FUNCTION_BLOCK farbzuordnung (* Basic Function Block Type *)
  (* Standard: 61499-2 *)
  (* Version 0.0, 19/08/2021, SESA56976, Schneider Electric, Template *)
  PACKAGE Main;
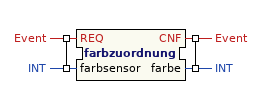
  EVENT_INPUT
    REQ WITH farbsensor; (* Normal Execution Request *)
  END_EVENT
  EVENT_OUTPUT
    CNF WITH farbe; (* Execution Confirmation *)
  END_EVENT
  VAR_INPUT
    farbsensor : INT; (* Input event qualifier *)
  END_VAR
  VAR_OUTPUT
    farbe : INT; (* Output event qualifier *)
  END_VAR
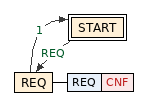
  EC_STATES
    START; (* Initial State *)
    REQ : REQ -> CNF; (* Normal execution *)
  END_STATES
  EC_TRANSITIONS
    START TO REQ := REQ;
    REQ TO START := 1;
  END_TRANSITIONS
  ALGORITHM REQ IN ST: (* Normally executed algorithm *)
IF  farbsensor <1000
THEN
farbe := 0;
END_IF;

IF  farbsensor > 1000 AND farbsensor <2000
THEN
farbe := 1;
END_IF;

IF  farbsensor > 2000 AND farbsensor <3000
THEN
farbe := 2;
END_IF;
  END_ALGORITHM
END_FUNCTION_BLOCK
